// TwinCAT 3 PLC project PRG_B_TestSupport
// Title: B_TestSupport
// Company: RafałOS
// Author: Rafał Osajda
// ProjectVersion: 0.0.0.1
// ProgramVersion: 3.1.4024.0
// libraries:
//   B_Base, * (RafalOS)
//   B_Base_HMI_Connector, * (RafalOS)
//   Tc2_Standard, * (Beckhoff Automation GmbH)
//   Tc2_System, * (Beckhoff Automation GmbH)
//   Tc3_Module, * (Beckhoff Automation GmbH)
// project tree:
//   DUTs/ ST_Components.TcDUT, ST_Components_HMI_Command.TcDUT, ST_Components_HMI_View.TcDUT, ST_ControlElements.TcDUT, ST_GroupElements.TcDUT, ST_TopElements.TcDUT
//   GVLs/ GVL_Elements.TcGVL, GVL_Variables.TcGVL
//   / PlcTask.TcTTO
//   POUs Compilation/ PRG_Compilation.TcPOU
//   POUs/01a_Komponent1 Logika/ FB_Component1.TcPOU, ITF_Component1.TcIO, ITF_Component1_HMI_Connector.TcIO, ITF_Component1_HMI_Connector_Command.TcIO, ITF_Component1_HMI_Connector_View.TcIO, ITF_Component1_HMI_Init.TcIO
//   POUs/02a_Komponent2 Logika/ FB_Component2.TcPOU, ITF_Component2.TcIO, ITF_Component2_HMI_Connector.TcIO, ITF_Component2_HMI_Connector_Command.TcIO, ITF_Component2_HMI_Connector_View.TcIO, ITF_Component2_HMI_Init.TcIO
//   POUs/03a_ElementWykonawczy1 Logika/ FB_Control1.TcPOU, ITF_Control1.TcIO, ITF_Control1_HMI_Connector.TcIO, ITF_Control1_HMI_Connector_Command.TcIO, ITF_Control1_HMI_Connector_View.TcIO, ITF_Control1_HMI_Init.TcIO
//   POUs/04a_ElementWykonawczy2 Logika/ FB_Control2.TcPOU, ITF_Control2.TcIO, ITF_Control2_HMI_Connector.TcIO, ITF_Control2_HMI_Connector_Command.TcIO, ITF_Control2_HMI_Connector_View.TcIO, ITF_Control2_HMI_Init.TcIO
//   POUs/05a_ElementZłożony1 Logika/ FB_Group1.TcPOU, ITF_Group1.TcIO, ITF_Group1_HMI_Connector.TcIO, ITF_Group1_HMI_Connector_Command.TcIO, ITF_Group1_HMI_Connector_View.TcIO, ITF_Group1_HMI_Init.TcIO
//   POUs/06a_ElementZłożony2 Logika/ FB_Group2.TcPOU, ITF_Group2.TcIO, ITF_Group2_HMI_Connector.TcIO, ITF_Group2_HMI_Connector_Command.TcIO, ITF_Group2_HMI_Connector_View.TcIO, ITF_Group2_HMI_Init.TcIO
//   POUs/07a_ElementZłożony3 Logika/ FB_Group3.TcPOU, ITF_Group3.TcIO, ITF_Group3_HMI_Connector.TcIO, ITF_Group3_HMI_Connector_Command.TcIO, ITF_Group3_HMI_Connector_View.TcIO, ITF_Group3_HMI_Init.TcIO
//   POUs/08a_ElementBazowy1 Logika/ FB_TopElement1.TcPOU, ITF_TopElement1_HMI_Connector.TcIO, ITF_TopElement1.TcIO, ITF_TopElement1_HMI_Connector_Command.TcIO, ITF_TopElement1_HMI_Connector_View.TcIO, ITF_TopElement1_HMI_Init.TcIO
//   POUs/09a_ElementBazowy2 Logika/ FB_TopElement2.TcPOU, ITF_TopElement2.TcIO, ITF_TopElement2_HMI_Connector.TcIO, ITF_TopElement2_HMI_Connector_Command.TcIO, ITF_TopElement2_HMI_Connector_View.TcIO, ITF_TopElement2_HMI_Init.TcIO
// real-time tasks:
//   TASK PlcTask: cycle T#10ms, priority 20, ADS port 350

CONFIGURATION PRG_B_TestSupport
    RESOURCE PLC ON TwinCAT3
        TASK PlcTask(INTERVAL := T#10ms, PRIORITY := 20);
        PROGRAM PRG_Compilation WITH PlcTask : PRG_Compilation;
    END_RESOURCE
END_CONFIGURATION

// ---- DUTs/ST_Components.TcDUT
TYPE ST_Components :
STRUCT
	fbCom01_Con01_T01		: FB_Component1;
	fbCom02_Con01_T01		: FB_Component1;
	fbCom03_Con01_T01		: FB_Component2;
	fbCom01_T01				: FB_Component1;
	fbCom02_T01				: FB_Component1;
	
	
	
END_STRUCT
END_TYPE

// ---- DUTs/ST_Components_HMI_Command.TcDUT
TYPE ST_Components_HMI_Command :
STRUCT
END_STRUCT
END_TYPE

// ---- DUTs/ST_Components_HMI_View.TcDUT
TYPE ST_Components_HMI_View :
STRUCT
END_STRUCT
END_TYPE

// ---- DUTs/ST_ControlElements.TcDUT
TYPE ST_ControlElements :
STRUCT
	fbCon01_T01			: FB_Control1 (
							itfC1	:= GVL_Elements.stComponents.fbCom01_Con01_T01,
	                	    itfC2	:= GVL_Elements.stComponents.fbCom02_Con01_T01,
	                	    itfC3	:= GVL_Elements.stComponents.fbCom03_Con01_T01
						);
END_STRUCT
END_TYPE

// ---- DUTs/ST_GroupElements.TcDUT
TYPE ST_GroupElements :
STRUCT
	
	
END_STRUCT
END_TYPE

// ---- DUTs/ST_TopElements.TcDUT
TYPE ST_TopElements :
STRUCT
	fbT1_01					: FB_TopElement1 (
								itfCon1			:= GVL_Elements.stControl.fbCon01_T01,
	                            itfCom1			:= GVL_Elements.stComponents.fbCom01_T01,
	                            itfCom2			:= GVL_Elements.stComponents.fbCom02_T01
							);
END_STRUCT
END_TYPE

// ---- GVLs/GVL_Elements.TcGVL
{attribute 'qualified_only'}
VAR_GLOBAL
	stComponents			: ST_Components;
	stComponentsView		: ST_Components_HMI_View;
	stComponentsCmd			: ST_Components_HMI_Command;
	stControl				: ST_ControlElements;
	stGroup					: ST_GroupElements;
	stTop					: ST_TopElements;
END_VAR

// ---- GVLs/GVL_Variables.TcGVL
{attribute 'qualified_only'}
VAR_GLOBAL
END_VAR

// ---- POUs/01a_Komponent1 Logika/ITF_Component1.TcIO
INTERFACE ITF_Component1 EXTENDS ITF_BaseComponent

END_INTERFACE

// ---- POUs/01a_Komponent1 Logika/ITF_Component1_HMI_Connector.TcIO
(*			
	RafalOS
	Rafał Osajda		22.12.2025		TC 4024.66
	Interejs łączacy kilka 
*)
INTERFACE ITF_Component1_HMI_Connector EXTENDS 
	ITF_BaseComponent_HMI_Connector, ITF_Component1_HMI_Connector_View, ITF_Component1_HMI_Connector_Command

END_INTERFACE

// ---- POUs/01a_Komponent1 Logika/ITF_Component1_HMI_Connector_Command.TcIO
INTERFACE ITF_Component1_HMI_Connector_Command EXTENDS ITF_BaseComponent_HMI_Connector_Command

END_INTERFACE

// ---- POUs/01a_Komponent1 Logika/ITF_Component1_HMI_Connector_View.TcIO
INTERFACE ITF_Component1_HMI_Connector_View EXTENDS ITF_BaseComponent_HMI_Connector_View

END_INTERFACE

// ---- POUs/01a_Komponent1 Logika/ITF_Component1_HMI_Init.TcIO
(*			
	RafalOS
	Rafał Osajda		22.12.2025		TC 4024.66
	Interfejs służacy jedynie w init do przekazywania elementu do łącznika HMI nie powinien posiadać żadnych metod
*)
INTERFACE ITF_Component1_HMI_Init EXTENDS ITF_BaseComponent, ITF_Component1_HMI_Connector

END_INTERFACE

// ---- POUs/02a_Komponent2 Logika/ITF_Component2.TcIO
INTERFACE ITF_Component2 EXTENDS ITF_BaseComponent

END_INTERFACE

// ---- POUs/02a_Komponent2 Logika/ITF_Component2_HMI_Connector.TcIO
(*			
	RafalOS
	Rafał Osajda		22.12.2025		TC 4024.66
	Interejs łączacy kilka 
*)
INTERFACE ITF_Component2_HMI_Connector EXTENDS 
	ITF_BaseComponent_HMI_Connector, ITF_Component2_HMI_Connector_View, ITF_Component2_HMI_Connector_Command

END_INTERFACE

// ---- POUs/02a_Komponent2 Logika/ITF_Component2_HMI_Connector_Command.TcIO
INTERFACE ITF_Component2_HMI_Connector_Command EXTENDS ITF_BaseComponent_HMI_Connector_Command

END_INTERFACE

// ---- POUs/02a_Komponent2 Logika/ITF_Component2_HMI_Connector_View.TcIO
INTERFACE ITF_Component2_HMI_Connector_View EXTENDS ITF_BaseComponent_HMI_Connector_View

END_INTERFACE

// ---- POUs/02a_Komponent2 Logika/ITF_Component2_HMI_Init.TcIO
(*			
	RafalOS
	Rafał Osajda		22.12.2025		TC 4024.66
	Interfejs służacy jedynie w init do przekazywania elementu do łącznika HMI nie powinien posiadać żadnych metod
*)
INTERFACE ITF_Component2_HMI_Init EXTENDS ITF_BaseComponent, ITF_Component2_HMI_Connector

END_INTERFACE

// ---- POUs/03a_ElementWykonawczy1 Logika/ITF_Control1.TcIO
INTERFACE ITF_Control1 EXTENDS ITF_BaseControlElement

END_INTERFACE

// ---- POUs/03a_ElementWykonawczy1 Logika/ITF_Control1_HMI_Connector.TcIO
INTERFACE ITF_Control1_HMI_Connector EXTENDS 
	ITF_BaseControlElement_HMI_Connector, ITF_Control1_HMI_Connector_View, ITF_Control1_HMI_Connector_Command

END_INTERFACE

// ---- POUs/03a_ElementWykonawczy1 Logika/ITF_Control1_HMI_Connector_Command.TcIO
INTERFACE ITF_Control1_HMI_Connector_Command EXTENDS ITF_BaseControlElement_HMI_Connector_Command

END_INTERFACE

// ---- POUs/03a_ElementWykonawczy1 Logika/ITF_Control1_HMI_Connector_View.TcIO
INTERFACE ITF_Control1_HMI_Connector_View EXTENDS ITF_BaseControlElement_HMI_Connector_View

END_INTERFACE

// ---- POUs/03a_ElementWykonawczy1 Logika/ITF_Control1_HMI_Init.TcIO
INTERFACE ITF_Control1_HMI_Init EXTENDS ITF_BaseControlElement, ITF_Control1_HMI_Connector

END_INTERFACE

// ---- POUs/04a_ElementWykonawczy2 Logika/ITF_Control2.TcIO
INTERFACE ITF_Control2 EXTENDS ITF_BaseControlElement

END_INTERFACE

// ---- POUs/04a_ElementWykonawczy2 Logika/ITF_Control2_HMI_Connector.TcIO
INTERFACE ITF_Control2_HMI_Connector EXTENDS 
	ITF_BaseControlElement_HMI_Connector, ITF_Control2_HMI_Connector_View, ITF_Control2_HMI_Connector_Command

END_INTERFACE

// ---- POUs/04a_ElementWykonawczy2 Logika/ITF_Control2_HMI_Connector_Command.TcIO
INTERFACE ITF_Control2_HMI_Connector_Command EXTENDS ITF_BaseControlElement_HMI_Connector_Command

END_INTERFACE

// ---- POUs/04a_ElementWykonawczy2 Logika/ITF_Control2_HMI_Connector_View.TcIO
INTERFACE ITF_Control2_HMI_Connector_View EXTENDS ITF_BaseControlElement_HMI_Connector_View

END_INTERFACE

// ---- POUs/04a_ElementWykonawczy2 Logika/ITF_Control2_HMI_Init.TcIO
INTERFACE ITF_Control2_HMI_Init EXTENDS ITF_BaseControlElement, ITF_Control2_HMI_Connector

END_INTERFACE

// ---- POUs/05a_ElementZłożony1 Logika/ITF_Group1.TcIO
INTERFACE ITF_Group1 EXTENDS ITF_BaseGroupElement

END_INTERFACE

// ---- POUs/05a_ElementZłożony1 Logika/ITF_Group1_HMI_Connector.TcIO
INTERFACE ITF_Group1_HMI_Connector EXTENDS
	ITF_BaseGroupElement_HMI_Connector, ITF_Group1_HMI_Connector_View, ITF_Group1_HMI_Connector_Command

END_INTERFACE

// ---- POUs/05a_ElementZłożony1 Logika/ITF_Group1_HMI_Connector_Command.TcIO
INTERFACE ITF_Group1_HMI_Connector_Command EXTENDS ITF_BaseGroupElement_HMI_Connector_Command

END_INTERFACE

// ---- POUs/05a_ElementZłożony1 Logika/ITF_Group1_HMI_Connector_View.TcIO
INTERFACE ITF_Group1_HMI_Connector_View EXTENDS ITF_BaseGroupElement_HMI_Connector_View

END_INTERFACE

// ---- POUs/05a_ElementZłożony1 Logika/ITF_Group1_HMI_Init.TcIO
INTERFACE ITF_Group1_HMI_Init EXTENDS ITF_BaseGroupElement, ITF_Group1_HMI_Connector

END_INTERFACE

// ---- POUs/06a_ElementZłożony2 Logika/ITF_Group2.TcIO
INTERFACE ITF_Group2 EXTENDS ITF_BaseGroupElement

END_INTERFACE

// ---- POUs/06a_ElementZłożony2 Logika/ITF_Group2_HMI_Connector.TcIO
INTERFACE ITF_Group2_HMI_Connector EXTENDS
	ITF_BaseGroupElement_HMI_Connector, ITF_Group2_HMI_Connector_View, ITF_Group2_HMI_Connector_Command

END_INTERFACE

// ---- POUs/06a_ElementZłożony2 Logika/ITF_Group2_HMI_Connector_Command.TcIO
INTERFACE ITF_Group2_HMI_Connector_Command EXTENDS ITF_BaseGroupElement_HMI_Connector_Command

END_INTERFACE

// ---- POUs/06a_ElementZłożony2 Logika/ITF_Group2_HMI_Connector_View.TcIO
INTERFACE ITF_Group2_HMI_Connector_View EXTENDS ITF_BaseGroupElement_HMI_Connector_View

END_INTERFACE

// ---- POUs/06a_ElementZłożony2 Logika/ITF_Group2_HMI_Init.TcIO
INTERFACE ITF_Group2_HMI_Init EXTENDS ITF_BaseGroupElement, ITF_Group2_HMI_Connector

END_INTERFACE

// ---- POUs/07a_ElementZłożony3 Logika/ITF_Group3.TcIO
INTERFACE ITF_Group3 EXTENDS ITF_BaseGroupElement

END_INTERFACE

// ---- POUs/07a_ElementZłożony3 Logika/ITF_Group3_HMI_Connector.TcIO
INTERFACE ITF_Group3_HMI_Connector EXTENDS
	ITF_BaseGroupElement_HMI_Connector, ITF_Group3_HMI_Connector_View, ITF_Group3_HMI_Connector_Command

END_INTERFACE

// ---- POUs/07a_ElementZłożony3 Logika/ITF_Group3_HMI_Connector_Command.TcIO
INTERFACE ITF_Group3_HMI_Connector_Command EXTENDS ITF_BaseGroupElement_HMI_Connector_Command

END_INTERFACE

// ---- POUs/07a_ElementZłożony3 Logika/ITF_Group3_HMI_Connector_View.TcIO
INTERFACE ITF_Group3_HMI_Connector_View EXTENDS ITF_BaseGroupElement_HMI_Connector_View

END_INTERFACE

// ---- POUs/07a_ElementZłożony3 Logika/ITF_Group3_HMI_Init.TcIO
INTERFACE ITF_Group3_HMI_Init EXTENDS ITF_BaseGroupElement, ITF_Group3_HMI_Connector

END_INTERFACE

// ---- POUs/08a_ElementBazowy1 Logika/ITF_TopElement1_HMI_Connector.TcIO
INTERFACE ITF_TopElement1_HMI_Connector EXTENDS ITF_BaseTopElement_HMI_Connector,
	ITF_TopElement1_HMI_Connector_View, ITF_TopElement1_HMI_Connector_Command

END_INTERFACE

// ---- POUs/08a_ElementBazowy1 Logika/ITF_TopElement1.TcIO
INTERFACE ITF_TopElement1 EXTENDS ITF_BaseTopElement

END_INTERFACE

// ---- POUs/08a_ElementBazowy1 Logika/ITF_TopElement1_HMI_Connector_Command.TcIO
INTERFACE ITF_TopElement1_HMI_Connector_Command EXTENDS ITF_BaseTopElement_HMI_Connector_Command

END_INTERFACE

// ---- POUs/08a_ElementBazowy1 Logika/ITF_TopElement1_HMI_Connector_View.TcIO
INTERFACE ITF_TopElement1_HMI_Connector_View EXTENDS ITF_BaseTopElement_HMI_Connector_View

END_INTERFACE

// ---- POUs/08a_ElementBazowy1 Logika/ITF_TopElement1_HMI_Init.TcIO
INTERFACE ITF_TopElement1_HMI_Init EXTENDS ITF_BaseTopElement, ITF_TopElement1_HMI_Connector

END_INTERFACE

// ---- POUs/09a_ElementBazowy2 Logika/ITF_TopElement2.TcIO
INTERFACE ITF_TopElement2 EXTENDS ITF_BaseTopElement

END_INTERFACE

// ---- POUs/09a_ElementBazowy2 Logika/ITF_TopElement2_HMI_Connector.TcIO
INTERFACE ITF_TopElement2_HMI_Connector EXTENDS ITF_BaseTopElement_HMI_Connector,
	ITF_TopElement2_HMI_Connector_View, ITF_TopElement2_HMI_Connector_Command

END_INTERFACE

// ---- POUs/09a_ElementBazowy2 Logika/ITF_TopElement2_HMI_Connector_Command.TcIO
INTERFACE ITF_TopElement2_HMI_Connector_Command EXTENDS ITF_BaseTopElement_HMI_Connector_Command

END_INTERFACE

// ---- POUs/09a_ElementBazowy2 Logika/ITF_TopElement2_HMI_Connector_View.TcIO
INTERFACE ITF_TopElement2_HMI_Connector_View EXTENDS ITF_BaseTopElement_HMI_Connector_View

END_INTERFACE

// ---- POUs/09a_ElementBazowy2 Logika/ITF_TopElement2_HMI_Init.TcIO
INTERFACE ITF_TopElement2_HMI_Init EXTENDS ITF_BaseTopElement, ITF_TopElement2_HMI_Connector

END_INTERFACE

// ---- POUs Compilation/PRG_Compilation.TcPOU
PROGRAM PRG_Compilation
VAR
END_VAR

END_PROGRAM

// ---- POUs/01a_Komponent1 Logika/FB_Component1.TcPOU
FUNCTION_BLOCK FB_Component1 EXTENDS FB_BaseComponent IMPLEMENTS ITF_Component1, ITF_Component1_HMI_Connector
VAR
END_VAR

END_FUNCTION_BLOCK

// ---- POUs/02a_Komponent2 Logika/FB_Component2.TcPOU
FUNCTION_BLOCK FB_Component2 EXTENDS FB_BaseComponent IMPLEMENTS ITF_Component2, ITF_Component2_HMI_Connector
VAR
END_VAR

END_FUNCTION_BLOCK

// ---- POUs/03a_ElementWykonawczy1 Logika/FB_Control1.TcPOU
FUNCTION_BLOCK FB_Control1 EXTENDS FB_BaseControlElement IMPLEMENTS ITF_Control1, ITF_Control1_HMI_Connector
VAR
	itfCom1			: ITF_Component1;
	itfCom2			: ITF_Component1;
	itfCom3			: ITF_Component2;
END_VAR

METHOD FB_init : BOOL
VAR_INPUT
	bInitRetains : BOOL; // if TRUE, the retain variables are initialized (warm start / cold start)
	bInCopyCode : BOOL;  // if TRUE, the instance afterwards gets moved into the copy code (online change)
	itfC1			: ITF_Component1;
	itfC2			: ITF_Component1;
	itfC3			: ITF_Component2;
END_VAR
THIS^.itfCom1 := itfC1;
THIS^.SetText (eLocation := E_BaseLocation.pl, wsDescription := "Control 1 C1");
THIS^.SetText (eLocation := E_BaseLocation.en, wsDescription := "Control 1 C1");
THIS^.SetText (eLocation := E_BaseLocation.de, wsDescription := "Control 1 C1");
THIS^.itfCom1.SetName (stName := THIS^.GetTexts ());

THIS^.itfCom2 := itfC2;
THIS^.SetText (eLocation := E_BaseLocation.pl, wsDescription := "Control 1 C2");
THIS^.SetText (eLocation := E_BaseLocation.en, wsDescription := "Control 1 C2");
THIS^.SetText (eLocation := E_BaseLocation.de, wsDescription := "Control 1 C2");
THIS^.itfCom2.SetName (stName := THIS^.GetTexts ());

THIS^.itfCom3 := itfC3;
THIS^.SetText (eLocation := E_BaseLocation.pl, wsDescription := "Control 1 C3");
THIS^.SetText (eLocation := E_BaseLocation.en, wsDescription := "Control 1 C3");
THIS^.SetText (eLocation := E_BaseLocation.de, wsDescription := "Control 1 C3");
THIS^.itfCom3.SetName (stName := THIS^.GetTexts ());
END_METHOD

END_FUNCTION_BLOCK

// ---- POUs/04a_ElementWykonawczy2 Logika/FB_Control2.TcPOU
FUNCTION_BLOCK FB_Control2 EXTENDS FB_BaseControlElement IMPLEMENTS ITF_Control1, ITF_Control2_HMI_Connector
VAR
END_VAR

END_FUNCTION_BLOCK

// ---- POUs/05a_ElementZłożony1 Logika/FB_Group1.TcPOU
FUNCTION_BLOCK FB_Group1 EXTENDS FB_BaseGroupElement IMPLEMENTS ITF_Group1, ITF_Group1_HMI_Connector
VAR
END_VAR

END_FUNCTION_BLOCK

// ---- POUs/06a_ElementZłożony2 Logika/FB_Group2.TcPOU
FUNCTION_BLOCK FB_Group2 EXTENDS FB_BaseGroupElement IMPLEMENTS ITF_Group1, ITF_Group2_HMI_Connector
VAR
END_VAR

END_FUNCTION_BLOCK

// ---- POUs/07a_ElementZłożony3 Logika/FB_Group3.TcPOU
FUNCTION_BLOCK FB_Group3 EXTENDS FB_BaseGroupElement IMPLEMENTS ITF_Group1, ITF_Group3_HMI_Connector
VAR
END_VAR

END_FUNCTION_BLOCK

// ---- POUs/08a_ElementBazowy1 Logika/FB_TopElement1.TcPOU
FUNCTION_BLOCK FB_TopElement1 EXTENDS FB_BaseTopElement IMPLEMENTS ITF_TopElement1, ITF_TopElement1_HMI_Connector
VAR
	itfCon1				: ITF_Control1;
	itfCom1				: ITF_Component1;
	itfCom2				: ITF_Component1;
	

END_VAR

METHOD FB_init : BOOL
VAR_INPUT
	bInitRetains : BOOL; // if TRUE, the retain variables are initialized (warm start / cold start)
	bInCopyCode : BOOL;  // if TRUE, the instance afterwards gets moved into the copy code (online change)
	itfCon1				: ITF_Control1;
	itfCom1				: ITF_Component1;
	itfCom2				: ITF_Component1;
END_VAR
THIS^.itfCon1 := itfCon1;
THIS^.SetText (eLocation := E_BaseLocation.pl, wsDescription := "Control 1 T1");
THIS^.SetText (eLocation := E_BaseLocation.en, wsDescription := "Control 1 T1");
THIS^.SetText (eLocation := E_BaseLocation.de, wsDescription := "Control 1 T1");
THIS^.itfCon1.SetName (stName := THIS^.GetTexts ());

THIS^.itfCom1 := itfCom1;
THIS^.SetText (eLocation := E_BaseLocation.pl, wsDescription := "Component 1 T1");
THIS^.SetText (eLocation := E_BaseLocation.en, wsDescription := "Component 1 T1");
THIS^.SetText (eLocation := E_BaseLocation.de, wsDescription := "Component 1 T1");
THIS^.itfCom1.SetName (stName := THIS^.GetTexts ());

THIS^.itfCom2 := itfCom2;
THIS^.SetText (eLocation := E_BaseLocation.pl, wsDescription := "Component 2 T1");
THIS^.SetText (eLocation := E_BaseLocation.en, wsDescription := "Component 2 T1");
THIS^.SetText (eLocation := E_BaseLocation.de, wsDescription := "Component 2 T1");
THIS^.itfCom2.SetName (stName := THIS^.GetTexts ());
END_METHOD

END_FUNCTION_BLOCK

// ---- POUs/09a_ElementBazowy2 Logika/FB_TopElement2.TcPOU
FUNCTION_BLOCK FB_TopElement2 EXTENDS FB_BaseTopElement IMPLEMENTS ITF_TopElement1, ITF_TopElement2_HMI_Connector
VAR
	itfCon1				: ITF_Control1;
	itfCon2				: ITF_Control1;
	itfCom1				: ITF_Component1;
	

END_VAR

METHOD FB_init : BOOL
VAR_INPUT
	bInitRetains : BOOL; // if TRUE, the retain variables are initialized (warm start / cold start)
	bInCopyCode : BOOL;  // if TRUE, the instance afterwards gets moved into the copy code (online change)
	itfCon1				: ITF_Control1;
	itfCon2				: ITF_Control1;
	itfCom1				: ITF_Component1;
END_VAR
THIS^.itfCon1 := itfCon1;
THIS^.SetText (eLocation := E_BaseLocation.pl, wsDescription := "Control 1 T2");
THIS^.SetText (eLocation := E_BaseLocation.en, wsDescription := "Control 1 T2");
THIS^.SetText (eLocation := E_BaseLocation.de, wsDescription := "Control 1 T2");
THIS^.itfCon1.SetName (stName := THIS^.GetTexts ());

THIS^.itfCon2 := itfCon2;
THIS^.SetText (eLocation := E_BaseLocation.pl, wsDescription := "Control 2 T2");
THIS^.SetText (eLocation := E_BaseLocation.en, wsDescription := "Control 2 T2");
THIS^.SetText (eLocation := E_BaseLocation.de, wsDescription := "Control 2 T2");
THIS^.itfCon2.SetName (stName := THIS^.GetTexts ());

THIS^.itfCom1 := itfCom1;
THIS^.SetText (eLocation := E_BaseLocation.pl, wsDescription := "Component 1 T2");
THIS^.SetText (eLocation := E_BaseLocation.en, wsDescription := "Component 1 T2");
THIS^.SetText (eLocation := E_BaseLocation.de, wsDescription := "Component 1 T2");
THIS^.itfCom1.SetName (stName := THIS^.GetTexts ());
END_METHOD

END_FUNCTION_BLOCK
